// TIA Portal V20 export
TYPE "LKinCtrl_typePnPTrackingProperties"
   STRUCT
      active : Bool;   // TRUE: Tracking is active
      velocity : LReal;   // Velocity of OCS
      frame : "LKinCtrl_typeFrame";   // Base frame of OCS
      objectPosition : "LKinCtrl_typeFrame";   // Relative OCS shift in base frame
   END_STRUCT;
END_TYPE
